{attribute 'GeneratedUsingTerminal: IMecat-0007-0001'}
{attribute addProperty BoxType "IMecat-0007-0001"}
{attribute addProperty Id "Pdo_EntryAT %I*ARRAY[0..131] OF USINT132"}
{attribute addProperty CRC "2170192396"}
{attribute addProperty Size "132"}
TYPE DI_TxPDO_Map_DF955083 EXTENDS TcoIo.InputBase_8311D824 :
STRUCT
	{attribute addProperty Name "Pdo_Entry"}
	Pdo_Entry AT %I* : ARRAY[0..131] OF USINT;
END_STRUCT
END_TYPE

(* stored: Version 1.2.0.0, ProductVersion 3.1.4024.11
   DUT DI_TxPDO_Map_DF955083: Id {f53569b9-76fb-00f0-00e4-9550dd7edb9a} *)
